(* IEC 61131-3 sources: stickle/source, 2 files *)

(* ---- clampandsaw.st ---- *)
TYPE State : (
    AllStopped,
    ClampsExtending,
    ClampsExtended,
    SawExtending,
    SawExtended,
    SawRetracting,
    SawRetracted,
    ClampsRetracting,
    ClampsRetracted,
);
END_TYPE

{network_publish := 'PublishOnly'}
VAR_GLOBAL
    currentState: State := AllStopped;
    THNTD: BOOL := FALSE;
    reset: BOOL := FALSE;
    testString: STRING[256];
END_VAR

FUNCTION main : DINT //the main entrypoint must be a function, not a program. Otherwise, timers will cause segfaults
    PRG_ClampAndSaw();
END_FUNCTION

PROGRAM PRG_ClampAndSaw
    VAR
        stateMachine: FB_ClampAndSaw;
    END_VAR

    stateMachine();
END_PROGRAM

FUNCTION_BLOCK FB_ClampAndSaw
    VAR
        threeseconds: TON; //timers can only be referenced by Programs or other Function Blocks
    END_VAR

    VAR_EXTERNAL
        currentState: State;
        THNTD: BOOL;
        reset: BOOL;
    END_VAR

    IF reset THEN
        reset := false;
        currentState := AllStopped;
        RETURN;
    END_IF;

    CASE currentState OF
        AllStopped:
            IF THNTD THEN
                currentState := ClampsExtending;
            END_IF;

        ClampsExtending:
            currentState := ClampsExtended;

        ClampsExtended:
            currentState := SawExtending;

        SawExtending:
            currentState := SawExtended;

        SawExtended:
            threeseconds(IN:=TRUE, PT:=T#3s);

            IF threeseconds.Q THEN
                threeseconds(IN:=FALSE, PT:=T#3s);
                currentState := SawRetracting;
            END_IF;

        SawRetracting:
            currentState := SawRetracted;

        SawRetracted:
            currentState := ClampsRetracting;

        ClampsRetracting:
            currentState := ClampsRetracted;

        ClampsRetracted:
            currentState := AllStopped;
    END_CASE;
END_FUNCTION_BLOCK

FUNCTION GetState : DINT
    VAR_EXTERNAL
        currentState: State;
    END_VAR

    GetState := currentState;
END_FUNCTION

FUNCTION SetThntd
    VAR_INPUT
        input: BOOL;
    END_VAR

    VAR_EXTERNAL
        THNTD: BOOL;
    END_VAR

    THNTD := input;
END_FUNCTION

FUNCTION ResetState
    VAR_EXTERNAL
        reset: BOOL;
    END_VAR

    reset:=TRUE;
END_FUNCTION

(* ---- testallbuiltins.st ---- *)
TYPE XmlTestStruct
    : STRUCT
        Count: INT;
        Flag: BOOL;
        Label: STRING[16];
        Samples: ARRAY[0..3] OF DINT;
    END_STRUCT
END_TYPE

TYPE XmlTestGrid : ARRAY[0..1, 1..3] OF INT; END_TYPE

TYPE XmlTestAlias : DINT; END_TYPE

PROGRAM TestAllBuiltins
    VAR_EXTERNAL
        _PLC_OptSerialErrSta: ARRAY[1..2] OF _sOPTSERIALERR_STA;
        _PowerOnCount: UDINT;
        _PowerOnHour: UDINT;
        _Card1PowerFail: BOOL;
        _Card1PrgTransferCmd: _sPRGTRANSFER_CMD;
        _DeviceOutHoldCfg: WORD;
        _EC_StatisticsLogCycleSec: UINT;
        _EC_StatisticsLogEnable: BOOL;
        _EIP_TDLinkStartCmd: BOOL;
        _EIP_TDLinkStopCmd: BOOL;
        _EIP1_TDLinkStartCmd: BOOL;
        _EIP1_TDLinkStopCmd: BOOL;
    END_VAR

    VAR
        time1: TIME;
        usint1: USINT;
        info1: UINT;
        dateandtime1: DATE_AND_TIME;
        bool1: BOOL;
        uint1: UINT;
        dword1: DWORD;
        udint1: UDINT;
        string1: STRING;
        sid1: _sNXUNIT_ID;
        test1: _sOPTSERIALERR_STA;
        sizedString1: STRING[32];
        struct1: XmlTestStruct;
        grid1: XmlTestGrid;
        alias1: XmlTestAlias;
    END_VAR

    //builtin functions
    TraceSamp(usint1, usint1);
    TraceTrig(usint1);
    GetTraceStatus(usint1, bool1, bool1, bool1, bool1);
    SetAlarm(5, info1, info1);
    ResetAlarm(5);
    GetAlarm(uint1, uint1);
    GetPLCError(uint1, dword1);
    GetEIPError(uint1, dword1);
    GetMCError(uint1, dword1);
    GetECError(uint1, dword1);
    SetInfo(5, info1, info1);
    GetNTPStatus(dateandtime1, bool1);
    GetMyTaskStatus(time1, time1, time1, udint1, bool1, udint1);
    GetMyTaskInterval();
    Task_IsActive(string1);
    Lock(usint1);
    Unlock(usint1);
    ActEventTask(string1);
    Get10msClk();
    Get10msCnt();
    GetPrgHashCode(dword1, dword1, dword1, dword1);
END_PROGRAM
